	FUNCTION_BLOCK FB 399
	TITLE =G299M RECYCLING AIR FLAP KILN 2
	//COPYRIGHT:    (C) 2009  BUHLER AG, CH-9240 UZWIL, SWITZERLAND
	//
	//PRODUCT:      WinCoS_BIW01_09
	//
	//TITLE:        RECYCLING AIR FLAP KILN 2
	//                Machine group control
	//                Maschinengruppensteuerung
	//
	//--------------------------------------------------------------------------------
	//
	//IDENT:        AUTHOR:             DEPT:                              DATE:
	//
	//P01_FB399.1.0 K.Renz              CSB41                              08.Okt.2009
	//             1st Release
	//
	//--------------------------------------------------------------------------------
	//
	//PURPOSE:
	//
	//MANUAL :
	//
	//RESTRICTIONS:
	//
	//--------------------------------------------------------------------------------
	AUTHOR  : KR
	FAMILY  : USW
	VERSION : 9.9


	VAR
	  Gr       : FB10;	//Standard interface to group
	  InOutValue1    : DINT; //Data for user
	  InOutValue2    : DINT; //Data for user
	  OutWayConflict : BOOL;	//Data for user
	  OutSelectionOk : BOOL;	//Data for user
	  CmdNewValue : BOOL;	//Data for user
	  CmdNewJob   : BOOL;	//Data for user
	  OutCodeOK   : BOOL;	//Data for user
	  InEndOfJob  : BOOL ;	//Data for user
	  staWayOk      : BOOL ;	//Data for user
	  EdgeStartRelease : BOOL ;	//Data for user
	  USW8  : BOOL;	//Data for user
	  USW9 : BOOL;	//Data for user
	  USW10: BOOL;	//Data for user
	  USW11: BOOL;	//Data for user
	  USW12: BOOL;	//Data for user
	  USW13: BOOL;	//Data for user
	  USW14: BOOL;	//Data for user
	  USW15: BOOL;	//Data for user
	     #A_3235_MXZ11I1 : FB14;   // DigInpCont
	     #A_3235_MXZ11I2 : FB14;   // DigInpCont
	     #A_3235_MXZ11 : FB20;   // VLS4Ctrl
	     #A_3236_MXZ11I1 : FB14;   // DigInpCont
	     #A_3236_MXZ11I2 : FB14;   // DigInpCont
	     #A_3236_MXZ11 : FB20;   // VLS4Ctrl
	     spare316 : ARRAY[316..571] of BYTE;
	     #A_3235_MXZ11I11 : FB14;   // DigInpCont
	     #A_3235_MXZ11I22 : FB14;   // DigInpCont
	     #A_3236_MXZ11I11 : FB14;   // DigInpCont
	     #A_3236_MXZ11I22 : FB14;   // DigInpCont
	END_VAR
	VAR_TEMP
	   tmpEnable		: BOOL;
	   tmpFlag  		: BOOL;
	   tmpCmdNext		: BOOL;
	   tmpLocal  		: BOOL;
	   tmpAspOk  		: BOOL;
	   tmpHWStop 		: BOOL;
	   tmpInstanzDBNo       : INT ;
	END_VAR
	BEGIN
	NETWORK
	TITLE =
	NETWORK
	TITLE =Read command from group control
	//Parameter
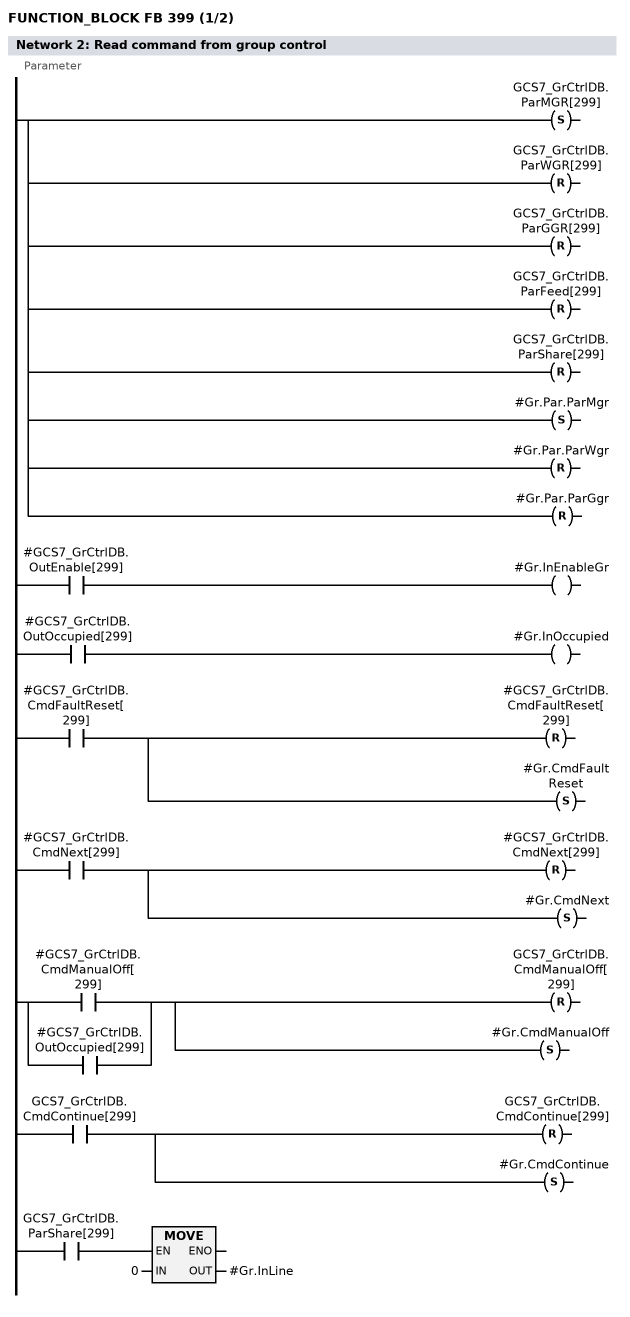
	      SET;
	      S   GCS7_GrCtrlDB.ParMGR[299];
	      R   GCS7_GrCtrlDB.ParWGR[299];
	      R   GCS7_GrCtrlDB.ParGGR[299];
	      R   GCS7_GrCtrlDB.ParFeed[299];
	      R   GCS7_GrCtrlDB.ParShare[299];
	      S   #Gr.Par.ParMgr;
	      R   #Gr.Par.ParWgr;
	      R   #Gr.Par.ParGgr;
	//Command
	      U   #GCS7_GrCtrlDB.OutEnable[299];
	      =   #Gr.InEnableGr;
	      U   #GCS7_GrCtrlDB.OutOccupied[299];
	      =   #Gr.InOccupied;
	      U   #GCS7_GrCtrlDB.CmdFaultReset[299];
	      R   #GCS7_GrCtrlDB.CmdFaultReset[299];
	      S   #Gr.CmdFaultReset;
	      U  #GCS7_GrCtrlDB.CmdNext[299];
	      R   #GCS7_GrCtrlDB.CmdNext[299];
	      S   #Gr.CmdNext;
	      U   #GCS7_GrCtrlDB.CmdManualOff[299];
	      O   #GCS7_GrCtrlDB.OutOccupied[299];
	      R   GCS7_GrCtrlDB.CmdManualOff[299];
	      S   #Gr.CmdManualOff;
	      U  GCS7_GrCtrlDB.CmdContinue[299];
	      R   GCS7_GrCtrlDB.CmdContinue[299];
	      S   #Gr.CmdContinue;
	//Init Line Number
	      U   GCS7_GrCtrlDB.ParShare[299];
	      SPBN WE00;
	      L     0;
	      T     #Gr.InLine;
	WE00: NOP   0;
	NETWORK
	TITLE =Call Methode Control
	// 1. Handle Interface PCControl
	// 2. Prepare mode --> ModePassive,ModeActive,ModeIdling
	// 3. Reset global flags of the group
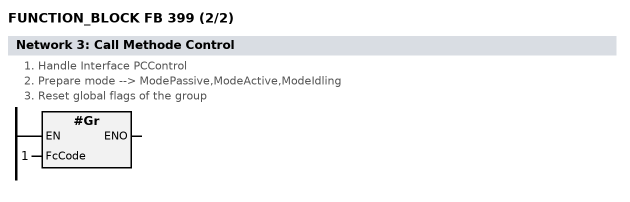
	      CALL #Gr (
	           FcCode                   := 1);
	NETWORK
	TITLE =Restart Idling Time
		L  #Gr.Par.ParIdling;
		L  2;
		>=I;
		SPB IdTm;
		T  #Gr.Par.ParIdling;
	IdTm:   NOP 0;
	      CLR;
	      S    #Gr.CmdRestartIdling;
	NETWORK
	TITLE =Prepare global flags
	NETWORK
	TITLE =Set Pattern (Target position)
	NETWORK
	TITLE =Interlocking WayOk
	//
	NETWORK
	TITLE =Interlocking Autostart
		CLR;
		R   #Gr.OutAutostart;
	NETWORK
	TITLE =Interlocking Enable
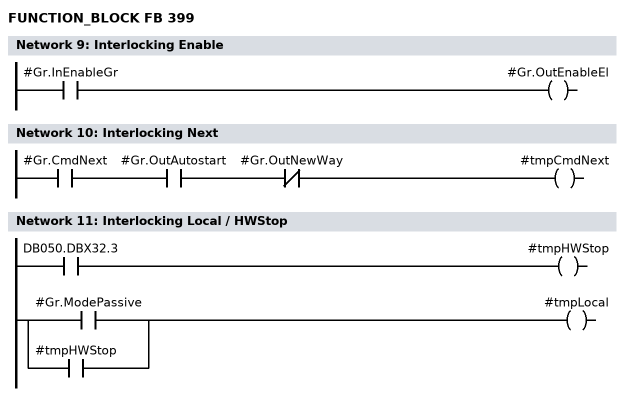
	      U     #Gr.InEnableGr;
	      =     #Gr.OutEnableEl;

	NETWORK
	TITLE =Interlocking Next
	      U     #Gr.CmdNext;
	      U     #Gr.OutAutostart;
	      UN    #Gr.OutNewWay;
	      =    #tmpCmdNext;

	NETWORK
	TITLE =Interlocking Local / HWStop
	      U    DB050.DBX32.3;
	      =    #tmpHWStop;

	      U    #Gr.ModePassive;
	      O    #tmpHWStop;
	      =    #tmpLocal;

	NETWORK
	TITLE ==A-3235-MXZ11I1 : LOUVER RECYCLE AIR 1 CLOSING
	NOP 0;
	//-InLocal---
	      U     #tmpLocal;
	      =     #A_3235_MXZ11I1.InLocal;
	//
	//-Monitoring---
	      SET;
	      =      #A_3235_MXZ11I1.InMonTrue;
	      CLR;
	      =      #A_3235_MXZ11I1.InMonFalse;
	//
	//-PreAlarm---
	      CLR;
	      =      #A_3235_MXZ11I1.InPreAlarmTrue;
	      CLR;
	      =      #A_3235_MXZ11I1.InPreAlarmFalse;
	//
	//-Additional commands---
	//      CLR
	//      S     #A_3235_MXZ11I1.CmdRunTimeOutTime
	//
	//-Read inputs---
	      U     E 1001.0;
	      =     #A_3235_MXZ11I1.InpTrue;
	      U   DB050.DBX32.4;
	      =     #A_3235_MXZ11I1.InHWStop;
	       U     PLC_DPInfo.Master[1].SlavesError[101];
	       =       #A_3235_MXZ11I1.InDPFault;
	//
	//-Set Parameters---
	//
	//-Call object control---
	      CALL  #A_3235_MXZ11I1;
	//
	//-Write outputs---
	NETWORK
	TITLE ==A-3235-MXZ11I2 : LOUVER RECYCLE AIR 1 OPENING
	NOP 0;
	//-InLocal---
	      U     #tmpLocal;
	      =     #A_3235_MXZ11I2.InLocal;
	//
	//-Monitoring---
	      SET;
	      =      #A_3235_MXZ11I2.InMonTrue;
	      CLR;
	      =      #A_3235_MXZ11I2.InMonFalse;
	//
	//-PreAlarm---
	      CLR;
	      =      #A_3235_MXZ11I2.InPreAlarmTrue;
	      CLR;
	      =      #A_3235_MXZ11I2.InPreAlarmFalse;
	//
	//-Additional commands---
	//      CLR
	//      S     #A_3235_MXZ11I2.CmdRunTimeOutTime
	//
	//-Read inputs---
	      U     E 1001.1;
	      =     #A_3235_MXZ11I2.InpTrue;
	      U   DB050.DBX32.4;
	      =     #A_3235_MXZ11I2.InHWStop;
	       U     PLC_DPInfo.Master[1].SlavesError[101];
	       =       #A_3235_MXZ11I2.InDPFault;
	//
	//-Set Parameters---
	//
	//-Call object control---
	      CALL  #A_3235_MXZ11I2;
	//
	//-Write outputs---
	NETWORK
	TITLE ==A-3235-MXZ11 : LOUVER RECYCLE AIR 1
	NOP 0;
	//-InLocal---
	      U     #tmpLocal;
	      =     #A_3235_MXZ11.InLocal;
	//
	//-Interlocking---
	      UN     #Gr.OutEnableEl;
	      =     #A_3235_MXZ11.InLN;
	      U    #Gr.OutEnableEl;
	      S     #A_3235_MXZ11.CmdMiddle1;
	      S     #A_3235_MXZ11.CmdMiddle2;
	      S     #A_3235_MXZ11.CmdHN;
	//
	//-Read inputs---
	      U     E 1004.6;
	      =     #A_3235_MXZ11.InpLN;
	      CLR;
	      =     #A_3235_MXZ11.InpMiddle1;
	      U     E 1004.7;
	      =     #A_3235_MXZ11.InpHN;
	      U   DB050.DBX32.4;
	      =     #A_3235_MXZ11.InHWStop;
	       U     PLC_DPInfo.Master[1].SlavesError[101];
	       =       #A_3235_MXZ11.InDPFault;
	//
	//-Set Parameters---
	//
	//-Call object control---
	      CALL  #A_3235_MXZ11;
	//
	//-Write outputs---
	      U     #A_3235_MXZ11.OutpLN;
	      =     A 1001.0;
	      U     #A_3235_MXZ11.OutpHN;
	      =     A 1001.1;
	NETWORK
	TITLE ==A-3236-MXZ11I1 : LOUVER RECYCLE AIR 2 CLOSING
	NOP 0;
	//-InLocal---
	      U     #tmpLocal;
	      =     #A_3236_MXZ11I1.InLocal;
	//
	//-Monitoring---
	      SET;
	      =      #A_3236_MXZ11I1.InMonTrue;
	      CLR;
	      =      #A_3236_MXZ11I1.InMonFalse;
	//
	//-PreAlarm---
	      CLR;
	      =      #A_3236_MXZ11I1.InPreAlarmTrue;
	      CLR;
	      =      #A_3236_MXZ11I1.InPreAlarmFalse;
	//
	//-Additional commands---
	//      CLR
	//      S     #A_3236_MXZ11I1.CmdRunTimeOutTime
	//
	//-Read inputs---
	      U     E 1001.2;
	      =     #A_3236_MXZ11I1.InpTrue;
	      U   DB050.DBX32.4;
	      =     #A_3236_MXZ11I1.InHWStop;
	       U     PLC_DPInfo.Master[1].SlavesError[101];
	       =       #A_3236_MXZ11I1.InDPFault;
	//
	//-Set Parameters---
	//
	//-Call object control---
	      CALL  #A_3236_MXZ11I1;
	//
	//-Write outputs---
	NETWORK
	TITLE ==A-3236-MXZ11I2 : LOUVER RECYCLE AIR 2 OPENING
	NOP 0;
	//-InLocal---
	      U     #tmpLocal;
	      =     #A_3236_MXZ11I2.InLocal;
	//
	//-Monitoring---
	      SET;
	      =      #A_3236_MXZ11I2.InMonTrue;
	      CLR;
	      =      #A_3236_MXZ11I2.InMonFalse;
	//
	//-PreAlarm---
	      CLR;
	      =      #A_3236_MXZ11I2.InPreAlarmTrue;
	      CLR;
	      =      #A_3236_MXZ11I2.InPreAlarmFalse;
	//
	//-Additional commands---
	//      CLR
	//      S     #A_3236_MXZ11I2.CmdRunTimeOutTime
	//
	//-Read inputs---
	      U     E 1001.3;
	      =     #A_3236_MXZ11I2.InpTrue;
	      U   DB050.DBX32.4;
	      =     #A_3236_MXZ11I2.InHWStop;
	       U     PLC_DPInfo.Master[1].SlavesError[101];
	       =       #A_3236_MXZ11I2.InDPFault;
	//
	//-Set Parameters---
	//
	//-Call object control---
	      CALL  #A_3236_MXZ11I2;
	//
	//-Write outputs---
	NETWORK
	TITLE ==A-3236-MXZ11 : LOUVER RECYCLE AIR 2
	NOP 0;
	//-InLocal---
	      U     #tmpLocal;
	      =     #A_3236_MXZ11.InLocal;
	//
	//-Interlocking---
	      UN     #Gr.OutEnableEl;
	      =     #A_3236_MXZ11.InLN;
	      U    #Gr.OutEnableEl;
	      S     #A_3236_MXZ11.CmdMiddle1;
	      S     #A_3236_MXZ11.CmdMiddle2;
	      S     #A_3236_MXZ11.CmdHN;
	//
	//-Read inputs---
	      U     E 1005.0;
	      =     #A_3236_MXZ11.InpLN;
	      CLR;
	      =     #A_3236_MXZ11.InpMiddle1;
	      U     E 1005.1;
	      =     #A_3236_MXZ11.InpHN;
	      U   DB050.DBX32.4;
	      =     #A_3236_MXZ11.InHWStop;
	       U     PLC_DPInfo.Master[1].SlavesError[101];
	       =       #A_3236_MXZ11.InDPFault;
	//
	//-Set Parameters---
	//
	//-Call object control---
	      CALL  #A_3236_MXZ11;
	//
	//-Write outputs---
	      U     #A_3236_MXZ11.OutpLN;
	      =     A 1001.2;
	      U     #A_3236_MXZ11.OutpHN;
	      =     A 1001.3;
	NETWORK
	TITLE ==A-3235-MXZ11I11 : LOUVER RECYCLE AIR 1 CLOSED
	NOP 0;
	//-InLocal---
	      U     #tmpLocal;
	      =     #A_3235_MXZ11I11.InLocal;
	//
	//-Monitoring---
	      CLR;
	      =      #A_3235_MXZ11I11.InMonTrue;
	      CLR;
	      =      #A_3235_MXZ11I11.InMonFalse;
	//
	//-PreAlarm---
	      CLR;
	      =      #A_3235_MXZ11I11.InPreAlarmTrue;
	      CLR;
	      =      #A_3235_MXZ11I11.InPreAlarmFalse;
	//
	//-Additional commands---
	//      CLR
	//      S     #A_3235_MXZ11I11.CmdRunTimeOutTime
	//
	//-Read inputs---
	      U     E 1001.0;
	      =     #A_3235_MXZ11I11.InpTrue;
	      U   DB050.DBX32.4;
	      =     #A_3235_MXZ11I11.InHWStop;
	       U     PLC_DPInfo.Master[1].SlavesError[101];
	       =       #A_3235_MXZ11I11.InDPFault;
	//
	//-Set Parameters---
	//
	//-Call object control---
	      CALL  #A_3235_MXZ11I11;
	//
	//-Write outputs---
	NETWORK
	TITLE ==A-3235-MXZ11I22 : LOUVER RECYCLE AIR 1 OPENED
	NOP 0;
	//-InLocal---
	      U     #tmpLocal;
	      =     #A_3235_MXZ11I22.InLocal;
	//
	//-Monitoring---
	      CLR;
	      =      #A_3235_MXZ11I22.InMonTrue;
	      CLR;
	      =      #A_3235_MXZ11I22.InMonFalse;
	//
	//-PreAlarm---
	      CLR;
	      =      #A_3235_MXZ11I22.InPreAlarmTrue;
	      CLR;
	      =      #A_3235_MXZ11I22.InPreAlarmFalse;
	//
	//-Additional commands---
	//      CLR
	//      S     #A_3235_MXZ11I22.CmdRunTimeOutTime
	//
	//-Read inputs---
	      U     E 1001.1;
	      =     #A_3235_MXZ11I22.InpTrue;
	      U   DB050.DBX32.4;
	      =     #A_3235_MXZ11I22.InHWStop;
	       U     PLC_DPInfo.Master[1].SlavesError[101];
	       =       #A_3235_MXZ11I22.InDPFault;
	//
	//-Set Parameters---
	//
	//-Call object control---
	      CALL  #A_3235_MXZ11I22;
	//
	//-Write outputs---
	NETWORK
	TITLE ==A-3236-MXZ11I11 : LOUVER RECYCLE AIR 2 CLOSED
	NOP 0;
	//-InLocal---
	      U     #tmpLocal;
	      =     #A_3236_MXZ11I11.InLocal;
	//
	//-Monitoring---
	      CLR;
	      =      #A_3236_MXZ11I11.InMonTrue;
	      CLR;
	      =      #A_3236_MXZ11I11.InMonFalse;
	//
	//-PreAlarm---
	      CLR;
	      =      #A_3236_MXZ11I11.InPreAlarmTrue;
	      CLR;
	      =      #A_3236_MXZ11I11.InPreAlarmFalse;
	//
	//-Additional commands---
	//      CLR
	//      S     #A_3236_MXZ11I11.CmdRunTimeOutTime
	//
	//-Read inputs---
	      U     E 1001.2;
	      =     #A_3236_MXZ11I11.InpTrue;
	      U   DB050.DBX32.4;
	      =     #A_3236_MXZ11I11.InHWStop;
	       U     PLC_DPInfo.Master[1].SlavesError[101];
	       =       #A_3236_MXZ11I11.InDPFault;
	//
	//-Set Parameters---
	//
	//-Call object control---
	      CALL  #A_3236_MXZ11I11;
	//
	//-Write outputs---
	NETWORK
	TITLE ==A-3236-MXZ11I22 : LOUVER RECYCLE AIR 2 OPENED
	NOP 0;
	//-InLocal---
	      U     #tmpLocal;
	      =     #A_3236_MXZ11I22.InLocal;
	//
	//-Monitoring---
	      CLR;
	      =      #A_3236_MXZ11I22.InMonTrue;
	      CLR;
	      =      #A_3236_MXZ11I22.InMonFalse;
	//
	//-PreAlarm---
	      CLR;
	      =      #A_3236_MXZ11I22.InPreAlarmTrue;
	      CLR;
	      =      #A_3236_MXZ11I22.InPreAlarmFalse;
	//
	//-Additional commands---
	//      CLR
	//      S     #A_3236_MXZ11I22.CmdRunTimeOutTime
	//
	//-Read inputs---
	      U     E 1001.3;
	      =     #A_3236_MXZ11I22.InpTrue;
	      U   DB050.DBX32.4;
	      =     #A_3236_MXZ11I22.InHWStop;
	       U     PLC_DPInfo.Master[1].SlavesError[101];
	       =       #A_3236_MXZ11I22.InDPFault;
	//
	//-Set Parameters---
	//
	//-Call object control---
	      CALL  #A_3236_MXZ11I22;
	//
	//-Write outputs---
	NETWORK
	TITLE =Test Fault
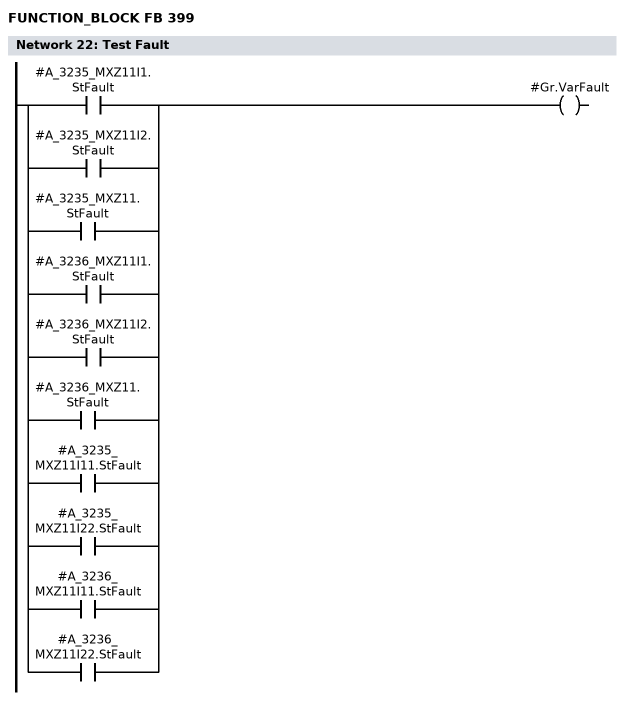
	      U     #A_3235_MXZ11I1.StFault;
	      O     #A_3235_MXZ11I2.StFault;
	      O     #A_3235_MXZ11.StFault;
	      O     #A_3236_MXZ11I1.StFault;
	      O     #A_3236_MXZ11I2.StFault;
	      O     #A_3236_MXZ11.StFault;
	      O     #A_3235_MXZ11I11.StFault;
	      O     #A_3235_MXZ11I22.StFault;
	      O     #A_3236_MXZ11I11.StFault;
	      O     #A_3236_MXZ11I22.StFault;
	      =     #Gr.VarFault;
	NETWORK
	TITLE =Test Warning
	      CLR;
	      =     #Gr.OutWarning;
	NETWORK
	TITLE =Test Stopped
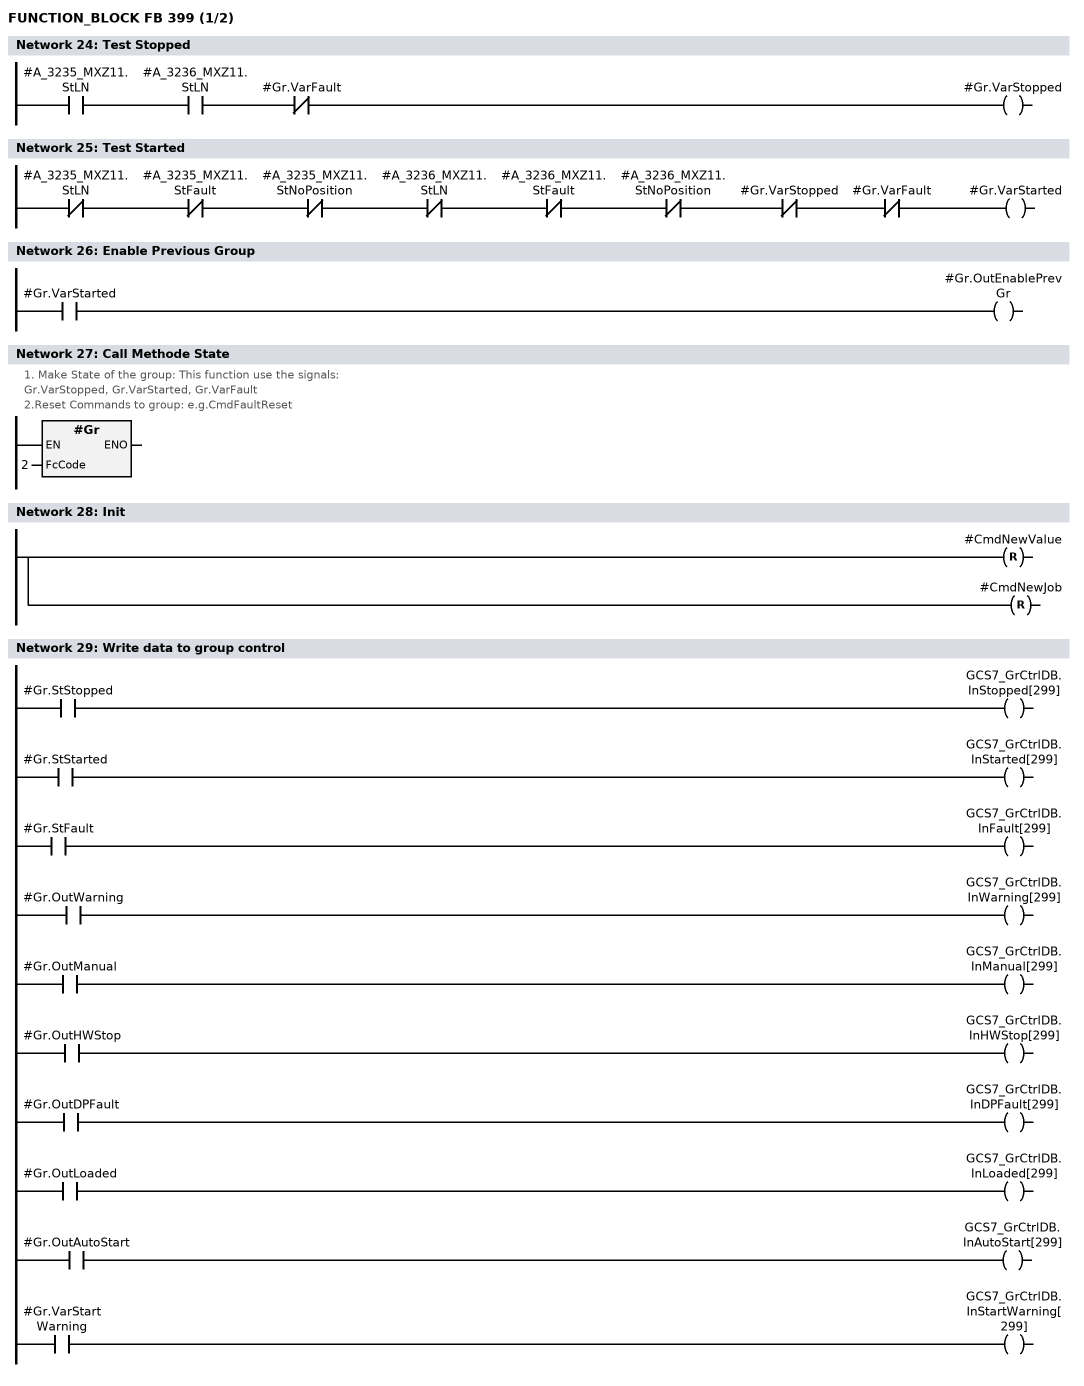
	      U     #A_3235_MXZ11.StLN;
	      U     #A_3236_MXZ11.StLN;
	      UN   #Gr.VarFault;
	      =     #Gr.VarStopped;
	NETWORK
	TITLE =Test Started
	      UN     #A_3235_MXZ11.StLN;
	      UN     #A_3235_MXZ11.StFault;
	      UN     #A_3235_MXZ11.StNoPosition;
	      UN     #A_3236_MXZ11.StLN;
	      UN     #A_3236_MXZ11.StFault;
	      UN     #A_3236_MXZ11.StNoPosition;
	      UN  #Gr.VarStopped;
	      UN  #Gr.VarFault;
	      =     #Gr.VarStarted;
	NETWORK
	TITLE =Enable Previous Group
	      U    #Gr.VarStarted;
	      =     #Gr.OutEnablePrevGr;
	NETWORK
	TITLE =Call Methode State
	//1. Make State of the group: This function use the signals:
	//        Gr.VarStopped, Gr.VarStarted, Gr.VarFault
	//2.Reset Commands to group: e.g.CmdFaultReset
	      CALL #Gr (
	           FcCode                   := 2);
	NETWORK
	TITLE =Init
	      SET;
	      R    #CmdNewValue;
	      R    #CmdNewJob;
	NETWORK
	TITLE =Write data to group control
	      U   #Gr.StStopped;
	      =   GCS7_GrCtrlDB.InStopped[299];
	      U   #Gr.StStarted;
	      =   GCS7_GrCtrlDB.InStarted[299];
	      U   #Gr.StFault;
	      =   GCS7_GrCtrlDB.InFault[299];
	      U   #Gr.OutWarning;
	      =   GCS7_GrCtrlDB.InWarning[299];
	      U   #Gr.OutManual;
	      =   GCS7_GrCtrlDB.InManual[299];
	      U   #Gr.OutHWStop;
	      =   GCS7_GrCtrlDB.InHWStop[299];
	      U   #Gr.OutDPFault;
	      =   GCS7_GrCtrlDB.InDPFault[299];
	      U   #Gr.OutLoaded;
	      =   GCS7_GrCtrlDB.InLoaded[299];
	      U   #Gr.OutAutoStart;
	      =   GCS7_GrCtrlDB.InAutoStart[299];
	      U   #Gr.VarStartWarning;
	      =   GCS7_GrCtrlDB.InStartWarning[299];
	NETWORK
	TITLE =End of block
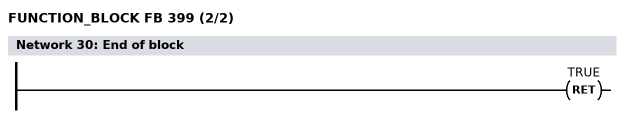

	BE

	END_FUNCTION_BLOCK
